{attribute 'linkalways'} 
{attribute 'no_explicit_call' := 'This FB is a CLASS and must be accessed using methods or properties'}
{attribute 'enable_dynamic_creation'}
FUNCTION_BLOCK Node_F_VN_LocateEdges EXTENDS VisionNode
VAR
	ipSrcImage : _ITcVnImage;
    ipEdgePoints : _ITcVnContainer;
    aStartPoint : _TcVnPoint2_REAL;
    aEndPoint : _TcVnPoint2_REAL;
    nNumEdges : _UDINT(0);
	eEdgeDirection : _ETcVnEdgeDirection(ETcVnEdgeDirection.TCVN_ED_DARK_TO_LIGHT);
    bAlternateDirection : _BOOL(FALSE);
    fMinStrength : _REAL(0.0);
    nSearchLines : _UDINT(1);
    hrPrev : _HRESULT(S_OK);
	hresult : _HRESULT(S_OK);
END_VAR

METHOD PUBLIC  Clone : I_Node
VAR
	pNode : POINTER TO Node_F_VN_LocateEdges;
END_VAR
pNode := __NEW(Node_F_VN_LocateEdges);
Clone := pNode^;
END_METHOD

METHOD FB_init : BOOL
VAR_INPUT
	bInitRetains : BOOL; // if TRUE, the retain variables are initialized (warm start / cold start)
	bInCopyCode : BOOL;  // if TRUE, the instance afterwards gets moved into the copy code (online change)
END_VAR
AddInput('ipSrcImage', ipSrcImage);
AddInput('aStartPoint', aStartPoint);
AddInput('aEndPoint', aEndPoint);
AddInput('hrPrev', hrPrev);
AddParameter('nNumEdges', nNumEdges);
AddParameter('eEdgeDirection', eEdgeDirection);
AddParameter('bAlternateDirection', bAlternateDirection);
AddParameter('fMinStrength', fMinStrength);
AddParameter('nSearchLines', nSearchLines);
AddOutput('ipEdgePoints', ipEdgePoints);
AddOutput('hresult',hresult);
END_METHOD

METHOD PROTECTED  OnExecute : HRESULT
hresult.Value := F_VN_LocateEdges(
	ipSrcImage := ipSrcImage.Value,
	ipEdgePoints := ipEdgePoints.Value,
    aStartPoint := aStartPoint.Value,
    aEndPoint := aEndPoint.Value,
    nNumEdges := nNumEdges.Value,
    eEdgeDirection := eEdgeDirection.Value,
    bAlternateDirection := bAlternateDirection.Value,
	fMinStrength := fMinStrength.Value,
	nSearchLines := nSearchLines.Value,
	hrPrev:= hrPrev.Value);
END_METHOD

METHOD PUBLIC PreExecutionCheck
VAR_INPUT
	Check : I_PreExecutionChecks;
END_VAR
IF FAILED(hrPrev.Value) THEN
    RETURN;
END_IF

Check.IsTrue(ipSrcImage.IsValid, 'ipSrcImage must contain an image');
Check.IsTrue(ipSrcImage.HasChannelCount(1), 'ipSrcImage must contain 1 channel');
Check.IsTrue(nSearchLines.IsOdd, 'nSearchLines must be an odd number');
END_METHOD

END_FUNCTION_BLOCK

(* stored: Version 1.1.0.1, ProductVersion 3.1.4024.13
   POU Node_F_VN_LocateEdges: Id {9b9932d8-46d2-033d-1562-615e0a37c130}, SpecialFunc None
   Folder Constructor: Id {02c50a26-c08b-04c2-005b-1ab263685286}
   Method Clone: Id {431c21b6-ca67-057e-15a2-0f466507243b}
   Method FB_init: Id {407891a7-66f6-0958-36fd-4f7a4f509719}
   Method OnExecute: Id {6f94ef24-40d7-03b0-1f76-94fbe57437ea}
   Method PreExecutionCheck: Id {66cc19c2-88b3-086b-1555-2eb405e70860} *)
